FUNCTION_BLOCK Gearbox (* Template for an empty basic function block *)
  (* Standard: 61499-2 *)
  (* Version 1.0, 2018-02-28, Duc Do Tran, OFFIS e.V. *)
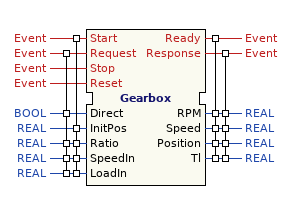
  EVENT_INPUT
    Start WITH Ratio, SpeedIn, InitPos, LoadIn;
    Request WITH Ratio, SpeedIn, LoadIn, Direct;
    Stop;
    Reset;
  END_EVENT
  EVENT_OUTPUT
    Ready WITH Speed, Position, RPM, Tl;
    Response WITH Speed, Position, RPM, Tl;
  END_EVENT
  VAR_INPUT
    Direct : BOOL;
    InitPos : REAL;
    Ratio : REAL;
    SpeedIn : REAL;
    LoadIn : REAL;
  END_VAR
  VAR_OUTPUT
    RPM : REAL;
    Speed : REAL;
    Position : REAL;
    Tl : REAL;
  END_VAR
  VAR
    bd : BOOL := TRUE; (* Internal Variable *)
    tg : REAL; (* Internal Variable *)
    phi : REAL; (* Internal Variable *)
    pi : REAL := 3.1415269; (* Internal Variable *)
    dphi : REAL; (* Internal Variable *)
    t0 : TIME; (* Internal Variable *)
    omega : REAL; (* Internal Variable *)
    temp : REAL; (* Internal Variable *)
  END_VAR
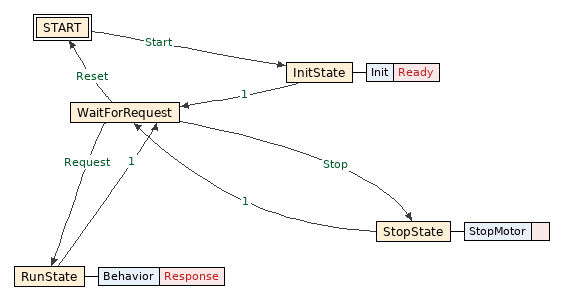
  EC_STATES
    START; (* Initial State *)
    RunState : Behavior -> Response;
    InitState : Init -> Ready;
    WaitForRequest;
    StopState : StopMotor;
  END_STATES
  EC_TRANSITIONS
    START TO InitState := Start;
    InitState TO WaitForRequest := 1;
    WaitForRequest TO RunState := Request;
    RunState TO WaitForRequest := 1;
    StopState TO WaitForRequest := 1;
    WaitForRequest TO StopState := Stop;
    WaitForRequest TO START := Reset;
  END_TRANSITIONS
  ALGORITHM Behavior IN ST: (* new algorithm *)
IF (bd = TRUE) THEN
	bd := FALSE;
	t0 := NOW_MONOTONIC();
END_IF;
omega := Ratio*SpeedIn;
Tl := Ratio*LoadIn;
tg := TIME_IN_S_TO_LREAL(NOW_MONOTONIC()-t0);
t0 := NOW_MONOTONIC();
dphi := omega*180*tg/pi;
phi := phi + dphi;
IF (Direct = TRUE) THEN // Run to LS2
	IF (phi >= 360) THEN
		phi := phi - 360;
	END_IF;
ELSE // Run to LS1
	IF (phi <= -360) THEN
		phi := phi + 360;
	END_IF;
END_IF;
Position := phi;
temp := omega*30/pi;
RPM := ABS(temp);
Speed := ABS(omega);
  END_ALGORITHM
  ALGORITHM Init IN ST: (* new algorithm *)
bd := TRUE;
Speed := 0;
IF (InitPos > 0) THEN
	IF (InitPos > 180) THEN
		phi :=180;
	ELSE
		phi := InitPos;
	END_IF;
ELSE
	phi := 0;
END_IF;
Position := phi;
  END_ALGORITHM
  ALGORITHM StopMotor IN ST: (* new algorithm *)
bd := TRUE;
Speed := 0;
  END_ALGORITHM
END_FUNCTION_BLOCK
